# EPICS IOC start-up script: output/git-repo/ts2-010crm_wtrc-plc-001/ts2_010crm_wtrc_plc_001-test-20220812164125.iocsh
#- @field MODVERSION
#- @runtime YES
#- The version of the PLC-IOC integration

#- @field ts2_010crm_wtrc_plc_001_VERSION
#- @runtime YES

#- Load plc interface database
dbLoadRecords("$(DBDIR=)ts2_010crm_wtrc_plc_001-test.db", "MODVERSION=$(PLCIOCVERSION)")
